FUNCTION_BLOCK AR2_TO_AR2IO (* Composite FB for convert AR2 to AR2IO *)
  (* Standard: 61499-2; Description: Copyright (c) 2024 HR Agrartechnik GmbH This program and the accompanying materials are made available under the terms of the Eclipse Public License 2.0 which is available at https://www.eclipse.org/legal/epl-2.0/ SPDX-License-Identifier: EPL-2.0 *)
  (* Version 1.0, 2024-04-24, Franz Höpfinger, HR Agrartechnik GmbH *)
  PACKAGE adapter::conversion::bidirectional;
  IMPORT eclipse4diac::core::TypeHash;
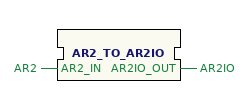
  SOCKETS
    AR2_IN : adapter::types::bidirectional::AR2; (* AR2 Adapter Input *)
  END_SOCKETS
  PLUGS
    AR2IO_OUT : adapter::types::bidirectional::AR2IO(D1 := 0.0); (* AR2IO Adapter Output *)
  END_PLUGS
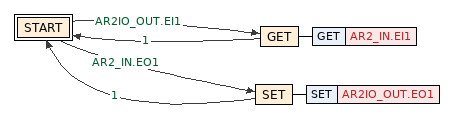
  EC_STATES
    START; (* Initial State *)
    GET : GET -> AR2_IN.EI1;
    SET : SET -> AR2IO_OUT.EO1;
  END_STATES
  EC_TRANSITIONS
    START TO GET := AR2IO_OUT.EI1;
    START TO SET := AR2_IN.EO1;
    GET TO START := 1;
    SET TO START := 1;
  END_TRANSITIONS
  ALGORITHM GET IN ST:
AR2_IN.DO1 := AR2IO_OUT.D1;
  END_ALGORITHM
  ALGORITHM SET IN ST:
AR2IO_OUT.D1 := AR2_IN.DI1;
  END_ALGORITHM
END_FUNCTION_BLOCK
